{attribute 'linkalways'} 
{attribute 'no_explicit_call' := 'This FB is a CLASS and must be accessed using methods or properties'}
{attribute 'enable_dynamic_creation'}
FUNCTION_BLOCK _TIMESTRUCT EXTENDS StructuredDatatypeBase
VAR
	localData : TIMESTRUCT;
	activeData : REFERENCE TO TIMESTRUCT REF= localData;
	_wYear : _WORD(localData.wYear);
	_wMonth : _WORD(localData.wMonth);
	_wDayOfWeek : _WORD(localData.wDayOfWeek);
	_wDay : _WORD(localData.wDay);
	_wHour : _WORD(localData.wHour);
	_wMinute : _WORD(localData.wMinute);
	_wSecond : _WORD(localData.wSecond);
	_wMilliseconds : _WORD(localData.wMilliseconds);
END_VAR

PROPERTY PUBLIC Address : PVOID
GET
Address := ADR(activeData);
END_GET
END_PROPERTY

METHOD PUBLIC ClearReference
VAR_INPUT
END_VAR
activeData REF= localData;
SetMemberReference();
END_METHOD

METHOD PUBLIC Clone : I_Datatype
VAR
    pClone : POINTER TO _TIMESTRUCT;
END_VAR
pClone := __NEW(_TIMESTRUCT());
pClone^.Value := Value;
Clone := pClone^;
END_METHOD

METHOD FB_init : BOOL
VAR_INPUT
	bInitRetains : BOOL; // if TRUE, the retain variables are initialized (warm start / cold start)
	bInCopyCode : BOOL;  // if TRUE, the instance afterwards gets moved into the copy code (online change)
END_VAR
SetMemberReference();
AddMember('wYear',_wYear);
AddMember('wMonth',_wMonth);
AddMember('wDayOfWeek',_wDayOfWeek);
AddMember('wDay',_wDay);
AddMember('wHour',_wHour);
AddMember('wMinute',_wMinute);
AddMember('wSecond',_wSecond);
AddMember('wMilliseconds',_wMilliseconds);
END_METHOD

PROPERTY PUBLIC Identifier : T_MAXSTRING
GET
Identifier := 'TIMESTRUCT';
END_GET
END_PROPERTY

METHOD PUBLIC MakeReferenceTo
VAR_INPUT
	ReferenceTarget : REFERENCE TO TIMESTRUCT;
END_VAR
activeData REF= ReferenceTarget;
SetMemberReference();
END_METHOD

METHOD PROTECTED SetMemberReference
VAR_INPUT
END_VAR
_wYear.MakeReferenceTo(activeData.wYear);
_wMonth.MakeReferenceTo(activeData.wMonth);
_wDayOfWeek.MakeReferenceTo(activeData.wDayOfWeek);
_wDay.MakeReferenceTo(activeData.wDay);
_wHour.MakeReferenceTo(activeData.wHour);
_wMinute.MakeReferenceTo(activeData.wMinute);
_wSecond.MakeReferenceTo(activeData.wSecond);
_wMilliseconds.MakeReferenceTo(activeData.wMilliseconds);
END_METHOD

PROPERTY PUBLIC Size : UDINT
GET
Size := SIZEOF(activeData);
END_GET
END_PROPERTY

METHOD TryMakeReferenceTo : BOOL
VAR_INPUT
	Target : I_Datatype;
END_VAR
VAR
	pTargetData : POINTER TO TIMESTRUCT;
END_VAR
IF NOT (Target.Name = Name) THEN
	RETURN;
END_IF

pTargetData := Target.Address;
activeData REF= pTargetData^;
SetMemberReference();
TryMakeReferenceTo := TRUE;
END_METHOD

PROPERTY PUBLIC Value : TIMESTRUCT
GET
Value := activeData;
END_GET
SET
activeData := Value;
END_SET
END_PROPERTY

PROPERTY PUBLIC wDay : Reference to _WORD
GET
wDay REF= _wDay;
END_GET
END_PROPERTY

PROPERTY PUBLIC wDayOfWeek : Reference to _WORD
GET
wDayOfWeek REF= _wDayOfWeek;
END_GET
END_PROPERTY

PROPERTY PUBLIC wHour : Reference to _WORD
GET
wHour REF= _wHour;
END_GET
END_PROPERTY

PROPERTY PUBLIC wMilliseconds : Reference to _WORD
GET
wMilliseconds REF= _wMilliseconds;
END_GET
END_PROPERTY

PROPERTY PUBLIC wMinute : Reference to _WORD
GET
wMinute REF= _wMinute;
END_GET
END_PROPERTY

PROPERTY PUBLIC wMonth : Reference to _WORD
GET
wMonth REF= _wMonth;
END_GET
END_PROPERTY

PROPERTY PUBLIC wSecond : Reference to _WORD
GET
wSecond REF= _wSecond;
END_GET
END_PROPERTY

PROPERTY PUBLIC wYear : Reference to _WORD
GET
wYear REF= _wYear;
END_GET
END_PROPERTY

END_FUNCTION_BLOCK

(* stored: Version 1.1.0.1, ProductVersion 3.1.4024.12
   POU _TIMESTRUCT: Id {5cd1ebb6-916e-047a-0935-4d7a058edb73}, SpecialFunc None
   Folder Constructor: Id {1edcb607-c80c-0b35-0f67-481a273f6a9f}
   Folder Protected: Id {00c26157-c9c3-0adc-1259-c265dc406398}
   Property Address: Id {028a70a0-bf15-08b9-02e0-df2513968418}
   Get Get: Id {d591990e-6370-0c5d-1bd6-4b74c023aa51}
   Method ClearReference: Id {9502f8c6-d240-0fb2-2cca-09e1ae67faf8}
   Method Clone: Id {8caec8a0-0505-0b53-10df-04db4aded8ba}
   Method FB_init: Id {6797cf26-94df-0a77-09d2-8470087346fe}
   Property Identifier: Id {8bbfe43b-001b-07ab-14f1-c18a7ddbe936}
   Get Get: Id {9b4727a2-c8e0-0b75-2bc8-2fd1558c3abc}
   Method MakeReferenceTo: Id {989d0c27-ba52-0b75-1735-0d80658b75a4}
   Method SetMemberReference: Id {ac8caeae-c74f-0b2e-1707-0f1fbc31df18}
   Property Size: Id {9898c282-10a1-070a-3393-87ae0429580e}
   Get Get: Id {edac4f8e-7b9d-0199-00d7-36888d9b907f}
   Method TryMakeReferenceTo: Id {fadfe40b-d2b0-0101-2d95-dab58245f6fa}
   Property Value: Id {1356e963-36fc-0c8a-1591-f9008e798d8c}
   Get Get: Id {e0e830a2-351d-0e1a-1ab6-a46b1c6b5468}
   Set Set: Id {078f43e0-ed0d-0da4-0e2d-611f4d3420c9}
   Property wDay: Id {044eb8e0-3bff-09fc-1a3a-6e30aba8644e}
   Get Get: Id {9642ada9-7110-04d5-272e-d115e46cccb9}
   Property wDayOfWeek: Id {0a14bded-de09-01bf-3579-25f62114630c}
   Get Get: Id {40f6f7fa-db3b-0178-0a0f-3eea911f9fdb}
   Property wHour: Id {28e501b1-532f-0c87-377e-e08f7717d792}
   Get Get: Id {bfc1bb70-7cd2-080a-3d2b-0ceddfd7cbaa}
   Property wMilliseconds: Id {224072f1-0c87-010d-1028-3765114a016a}
   Get Get: Id {17edd676-6496-0563-1c1a-57ab20bf7100}
   Property wMinute: Id {5767927c-f514-0589-218a-c7ccc86f0540}
   Get Get: Id {f7c0fc90-aa93-013d-2d4a-5d800e691b95}
   Property wMonth: Id {60dda2f1-9a77-0192-3004-428e642364eb}
   Get Get: Id {54b809ff-cb87-06cb-2bf4-ac3d9c7948ff}
   Property wSecond: Id {59f97060-f5ff-0787-3fdc-43d832a20409}
   Get Get: Id {df2082b5-805e-0a08-1d24-9f97f6cdd4f3}
   Property wYear: Id {be36cb92-0bc4-091a-0c6d-b9d979d2b47e}
   Get Get: Id {abcf1821-d1fd-0117-36ee-871795779c19} *)
